Staubli VAL3: onBackEvent.pgx

program onBackEvent(bool& x_bSave[])
  local num i
  local string l_sItem
  local string l_sInstruction
  local num l_nIndex
  local num j
  local num l_nChar
  local num l_nResult
  local InstrItem l_iInstr
  local string l_sPath
begin
  //
  // NB sEvent is the selected
  // element in the LIST
  //
  // get the item
  call prog:getItem(l_iInstr,nIndex)
  // find the instruction to load
  call saveData:getPathInstr(l_iInstr.sType,l_sPath)
  j=events:libLoad(l_sPath)
  delay(0)
  if j==0
    // cal the onInsert function
    call events:onInsert(l_iInstr.sData)
    // insert the item
    if l_iInstr.sData!=""
      call prog:insertItem(l_iInstr,nIndex)
      if nIndex>0
        call prog:deleteItem(nIndex+1,l_nResult)
      endIf
      x_bSave=true
      logMsg("[KERNEL] INTERFACE:Insert new item: "+l_sItem)
      i=size(saveData:sInstr)-1
    endIf
    call buildList()
    //
  else
    popUpMsg("Loading event "+l_sInstruction+" error CODE "+toString("",j))
  endIf
  //
end
